  def rq_current_pos_norm(gripper_socket="1"):
      pos_gripper = rq_current_pos(gripper_socket)
      pos_norm = gripper_to_norm(pos_gripper)
      return pos_norm
  end

  def gripper_to_norm(value_gripper):
      value_norm = (value_gripper / 255) * 100
      return floor(value_norm)
  end

  def norm_to_gripper(value_norm):
      value_gripper = (value_norm / 100) * 255
      return ceil(value_gripper)
  end

  def rq_get_position():
      return rq_current_pos_norm()
  end

  def rq_gripper_led_on(gripper_socket="1"):
      rq_set_var("LBP",0, gripper_socket)
  end

  def rq_gripper_led_off(gripper_socket="1"):
      rq_set_var("LBP",1, gripper_socket)
      rq_set_var("LRD",0, gripper_socket)
      rq_set_var("LBL",0, gripper_socket)
      rq_set_var("LGN",0, gripper_socket)
  end

  def rq_gripper_led_force_red(gripper_socket="1"):
      rq_set_var("LBP",1, gripper_socket)
      rq_set_var("LRD",1, gripper_socket)
      rq_set_var("LBL",0, gripper_socket)
      rq_set_var("LGN",0, gripper_socket)
  end

  def rq_gripper_led_force_blue(gripper_socket="1"):
      rq_set_var("LBP",1, gripper_socket)
      rq_set_var("LRD",0, gripper_socket)
      rq_set_var("LBL",1, gripper_socket)
      rq_set_var("LGN",0, gripper_socket)
  end

  def rq_gripper_led_force_green(gripper_socket="1"):
      rq_set_var("LBP",1, gripper_socket)
      rq_set_var("LRD",0, gripper_socket)
      rq_set_var("LBL",0, gripper_socket)
      rq_set_var("LGN",1, gripper_socket)
  end

  def rq_gripper_led_force_purple(gripper_socket="1"):
      rq_set_var("LBP",1, gripper_socket)
      rq_set_var("LRD",1, gripper_socket)
      rq_set_var("LBL",1, gripper_socket)
      rq_set_var("LGN",0, gripper_socket)
  end

  ############################################
  # mm/inches functions
  ############################################
  gripper_closed_norm = [100, 100, 100, 100]
  gripper_open_norm = [0, 0, 0, 0]
  gripper_closed_mm = [0, 0, 0, 0]
  gripper_open_mm = [50, 50, 50, 50]

  def rq_current_pos_mm(gripper_socket=1):
      pos_gripper = rq_current_pos(gripper_socket)
      pos_mm = gripper_to_mm(pos_gripper, gripper_socket)
      return round_value_2_dec(pos_mm)
  end

  def rq_current_pos_inches(gripper_socket=1):
      pos_gripper = rq_current_pos(gripper_socket)
      pos_mm = gripper_to_mm(pos_gripper, gripper_socket)
      pos_in = pos_mm / 25.4
      return round_value_2_dec(pos_in)
  end

  def rq_move_mm(pos_mm, gripper_socket=1):
      pos_gripper = mm_to_gripper(pos_mm, gripper_socket)
      rq_move(pos_gripper, gripper_socket)
  end

  def rq_move_and_wait_mm(pos_mm, gripper_socket=1):
      pos_gripper = mm_to_gripper(pos_mm, gripper_socket)
      rq_move_and_wait(pos_gripper, gripper_socket)
  end

  def rq_move_inches(pos_in, gripper_socket=1):
      pos_mm = pos_in * 25.4
      rq_move_mm(pos_mm, gripper_socket)
  end

  def rq_move_and_wait_inches(pos_in, gripper_socket=1):
      pos_mm = pos_in * 25.4
      rq_move_and_wait_mm(pos_mm, gripper_socket)
  end

  def get_closed_norm(gripper_socket):
      return gripper_closed_norm[gripper_socket - 1]
  end

  def get_open_norm(gripper_socket):
      return gripper_open_norm[gripper_socket - 1]
  end

  def get_closed_mm(gripper_socket):
      return gripper_closed_mm[gripper_socket - 1]
  end

  def get_open_mm(gripper_socket):
      return gripper_open_mm[gripper_socket - 1]
  end

  def set_closed_norm(closed_norm, gripper_socket):
      gripper_closed_norm[gripper_socket - 1] = closed_norm
  end

  def set_open_norm(open_norm, gripper_socket):
      gripper_open_norm[gripper_socket - 1] = open_norm
  end

  def set_closed_mm(closed_mm, gripper_socket):
      gripper_closed_mm[gripper_socket - 1] = closed_mm
  end

  def set_open_mm(open_mm, gripper_socket):
      gripper_open_mm[gripper_socket - 1] = open_mm
  end

  def gripper_to_mm(value_gripper, gripper_socket):
      closed_norm = get_closed_norm(gripper_socket)
      open_norm = get_open_norm(gripper_socket)
      closed_mm = get_closed_mm(gripper_socket)
      open_mm = get_open_mm(gripper_socket)

      value_norm = (value_gripper / 255) * 100

      slope = (closed_mm - open_mm) / (closed_norm - open_norm)
      value_mm = slope * (value_norm - closed_norm) + closed_mm

      if (value_mm > open_mm):
          value_mm_limited = open_mm
      elif (value_mm < closed_mm):
          value_mm_limited = closed_mm
      else:
          value_mm_limited = value_mm
      end

      return value_mm_limited
  end

  def mm_to_gripper(value_mm, gripper_socket):
      closed_norm = get_closed_norm(gripper_socket)
      open_norm = get_open_norm(gripper_socket)
      closed_mm = get_closed_mm(gripper_socket)
      open_mm = get_open_mm(gripper_socket)

      slope = (closed_norm - open_norm) / (closed_mm - open_mm)
      value_norm = (value_mm - closed_mm) * slope + closed_norm

      value_gripper = value_norm * 255 / 100

      if (value_gripper > 255):
          value_gripper_limited = 255
      elif (value_gripper < 0):
          value_gripper_limited = 0
      else:
          value_gripper_limited = round_value(value_gripper)
      end

      return value_gripper_limited
  end

  def round_value(value):
      value_mod = value % 1

      if(value_mod < 0.5):
          return floor(value)
      else:
          return ceil(value)
      end
  end

  def round_value_2_dec(value):
      value_x_100 = value * 100
      value_x_100_rounded = round_value(value_x_100)
      return value_x_100_rounded / 100
  end

  def clear_socket_buffer(gripper_socket="1", read_timeout = 0.1):
      rq_comm_clear_socket_buffer_enabled[rq_socket_to_index(gripper_socket)] = True
  end

  def rq_gripper_id_to_ascii(gripper_id):
      if(gripper_id == "1"):
          return 57
      elif(gripper_id == "2"):
          return 50
      elif(gripper_id == "3"):
          return 51
      elif(gripper_id == "4"):
          return 52
      end
  end

  def scale(value, rawRange, scaledRange):
      def computeSlope(inputRange, outputRange):
          outputRangeDelta = outputRange[1] - outputRange[0]
          inputRangeDelta = inputRange[1] - inputRange[0]

          if (inputRangeDelta == 0):
              return 0
          else:
              return outputRangeDelta / inputRangeDelta
          end
      end

      def computeIntercept(slope, inputRange, outputRange):
          return outputRange[0] - (slope * inputRange[0])
      end

      def clipScaledValue(outputScaledValue, outputRange):
          if (outputRange[0] < outputRange[1]):
              return clipWhenLowerLimitIsLessThanHigher(outputScaledValue, outputRange)
          else:
              return clipWhenLowerLimitIsGreaterThanHigherLimit(outputScaledValue, outputRange)
          end
      end

      def clipWhenLowerLimitIsGreaterThanHigherLimit(outputScaledValue, outputRange):
          if (outputScaledValue < outputRange[1]):
              return outputRange[1]
          elif (outputScaledValue > outputRange[0]):
              return outputRange[0]
          else:
              return outputScaledValue
          end
      end

      def clipWhenLowerLimitIsLessThanHigher(outputScaledValue, outputRange):
          if (outputScaledValue < outputRange[0]):
              return outputRange[0]
          elif (outputScaledValue > outputRange[1]):
              return outputRange[1]
          else:
              return outputScaledValue
          end
      end

      slope = computeSlope(rawRange, scaledRange)
      intercept = computeIntercept(slope, rawRange, scaledRange)
      scaledValue = slope * value + intercept
      return clipScaledValue(scaledValue, scaledRange)
  end

  def limit(value, range):
      return scale(value, range, range)
  end


  rq_init_comm_if_connected(9, "1")
  rq_init_comm_if_connected(2, "2")
  rq_init_comm_if_connected(3, "3")
  rq_init_comm_if_connected(4, "4")
  rq_print_connected_grippers()
  rq_gripper_communication_thread = run rq_gripper_communication()
  set_closed_norm(100.0, 1)
  set_open_norm(0.0, 1)
  set_closed_mm(0.0, 1)
  set_open_mm(50.0, 1)
  set_closed_norm(100.0, 2)
  set_open_norm(0.0, 2)
  set_closed_mm(0.0, 2)
  set_open_mm(50.0, 2)
  set_closed_norm(100.0, 3)
  set_open_norm(0.0, 3)
  set_closed_mm(0.0, 3)
  set_open_mm(50.0, 3)
  set_closed_norm(100.0, 4)
  set_open_norm(0.0, 4)
  set_closed_mm(0.0, 4)
  set_open_mm(50.0, 4)
  rq_current_limit_enabled = False
  while(not rq_gripper_communication_thread_started):
      sleep(0.008)
  end
  # end: URCap Installation Node
  global cnt_1=0
  global volo=0
  global volo_is_counting=False
  thread Timer_Thread():
    while (True):
      if (volo_is_counting):
        volo = volo + get_steptime()
      end
      sync()
    end
  end
  run Timer_Thread()
  while (True):
    $ 1 "Robot Program"
    # begin: URCap Program Node
    #   Source: Robotiq_Grippers, 1.8.9.14887, Robotiq Inc.
    #   Type: Gripper Activate
    $ 2 "Gripper Activate"

    kill rq_gripper_communication_thread
    rq_gripper_communication_thread_started = False
    rq_close_gripper_socket("1")
    rq_close_gripper_socket("2")
    rq_close_gripper_socket("3")
    rq_close_gripper_socket("4")

    rq_init_comm_if_connected(9, "1")
    rq_init_comm_if_connected(2, "2")
    rq_init_comm_if_connected(3, "3")
    rq_init_comm_if_connected(4, "4")
    rq_print_connected_grippers()
    rq_gripper_communication_thread = run rq_gripper_communication()

    while(not rq_gripper_communication_thread_started):
        sleep(0.008)
    end

    rq_set_max_current_for_all_grippers()

    reset_and_activate = False

    rq_activate_all_grippers(False)
    # end: URCap Program Node
    # begin: URCap Program Node
    #   Source: Robotiq_Grippers, 1.8.9.14887, Robotiq Inc.
    #   Type: Gripper
    $ 3 "Gripper Open (1)"
    if not(gripper_connected[0]):
      popup("Gripper 1 must be connected to run this program.", "No connection", False, True, True)
    end
    if not(rq_is_gripper_activated("1")):
      popup("Gripper 1 is not activated. Go to Installation tab > Gripper to activate it and run the program again.", "Not activated", False, True, True)
    end
    rq_set_pos_spd_for(0, 0, 0, "1")
    rq_wait_pos_spe_for_request(0, 0, 0, "1")
    rq_go_to("1")
    rq_wait("1")
    # end: URCap Program Node
    $ 4 "volo: Stop"
    volo_is_counting = False
    $ 5 "ready≔ False "
    global ready=  False
    $ 6 "engineon≔Nastro_ON"
    global engineon=get_standard_digital_out(0)
    $ 7 "engineon≔ False "
    global engineon=  False
    $ 8 "sensoreBasso≔FC_Start"
    global sensoreBasso=get_standard_digital_in(4)
    $ 9 "sensoreAlto≔FC_High"
    global sensoreAlto=get_standard_digital_in(6)
    $ 10 "sensoreStop≔FC_End"
    global sensoreStop=get_standard_digital_in(5)
    $ 11 "tempoVolo≔4000"
    global tempoVolo=4000
    $ 12 "Loop"
    while (True):
      $ 13 "If FC_Start== True "
      if (get_standard_digital_in(4)==  True  ):
        $ 14 "engineon≔ True "
        global engineon=  True
        $ 15 "Wait FC_Start=LO"
        while (get_standard_digital_in(4) == True):
          sync()
        end
      else:
        $ 16 "ElseIf FC_High== True "
        if (get_standard_digital_in(6)==  True  ):
          $ 17 "engineon≔ True "
          global engineon=  True
          $ 18 "Wait FC_High=LO"
          while (get_standard_digital_in(6) == True):
            sync()
          end
        else:
          $ 19 "ElseIf FC_End== True "
          if (get_standard_digital_in(5)==  True  ):
            $ 20 "engineon≔ False "
            global engineon=  False
            $ 21 "MoveL"
            $ 22 "Waypoint_1" "breakAfter"
            movel(p[-.381387685375, -.169307009528, .186364165479, .031229211360, 3.092074785863, -.049669567106], a=1.2, v=0.25)
            $ 23 "MoveL"
            $ 24 "Waypoint_2" "breakAfter"
            movel(p[-.373641097354, -.171322588210, .081624890856, .031253673923, 3.092083063402, -.049651173659], a=1.2, v=0.25)
            # begin: URCap Program Node
            #   Source: Robotiq_Grippers, 1.8.9.14887, Robotiq Inc.
            #   Type: Gripper
            $ 25 "Gripper Move51% (1)"
            if not(gripper_connected[0]):
              popup("Gripper 1 must be connected to run this program.", "No connection", False, True, True)
            end
            if not(rq_is_gripper_activated("1")):
              popup("Gripper 1 is not activated. Go to Installation tab > Gripper to activate it and run the program again.", "Not activated", False, True, True)
            end
            rq_set_pos_spd_for(131, 0, 0, "1")
            rq_wait_pos_spe_for_request(131, 0, 0, "1")
            rq_go_to("1")
            rq_wait("1")
            # end: URCap Program Node
            $ 26 "MoveL"
            $ 27 "Waypoint_3" "breakAfter"
            movel(p[-.370356696043, -.174547637783, .216862429798, .031961409927, 3.097477882431, -.043978030525], a=1.2, v=0.25)
            $ 28 "MoveL"
            $ 29 "Waypoint_4" "breakAfter"
            movel(p[-.134875456305, -.252278271452, .221726537061, .032070337176, 3.097477750080, -.043854214395], a=1.2, v=0.25)
            $ 30 "Pallet"
            cnt_1_x = cnt_1 % 2
            cnt_1_y = floor(cnt_1 / 2)
            pose_1 = interpolate_pose(interpolate_pose(p[-.089762363593, -.429151138960, .009188706301, .027577147014, 3.053416589493, -.032182313128], p[.031186609987, -.429171211043, .011085502208, .027611575133, 3.053453182137, -.032263865590], cnt_1_x/1), interpolate_pose(p[-.089761553552, -.366553516844, .009168617974, .027481938487, 3.053493094310, -.032138841944], p[.031156149702, -.364086955268, .011056827590, .027631286382, 3.053463713793, -.032250855705],cnt_1_x/1), cnt_1_y/1)
            if (cnt_1 >= 3):
              cnt_1 = 0
            else:
              cnt_1 = cnt_1 + 1
            end
            $ 37 "Approach_1" "noBreak"
            movel(pose_trans(pose_1, pose_trans(pose_inv(p[-.089755279794, -.366542025468, .202492381968, .027482330613, 3.053431155792, -.032206448903]),p[-.089781181398, -.366546626212, .202507837739, .027606886294, 3.053463920443, -.032300040654])), a=1.2, v=0.25)
            $ 38 "PatternPoint_1" "noBreak"
            movel(pose_1, a=1.2, v=0.25)
            $ 39 "Set" "noBreak"
            $ 40 "Wait volo>tempoVolo" "noBreak"
            while (not(volo>tempoVolo)):
              sync()
            end
            $ 41 "Exit_1" "noBreak"
            movel(pose_trans(pose_1, pose_trans(pose_inv(p[-.089755279794, -.366542025468, .202492381968, .027482330613, 3.053431155792, -.032206448903]),p[-.089763731108, -.366543702749, .202497776555, .027500770851, 3.053466015947, -.032225658991])), a=1.2, v=0.25)
            $ 42 "volo: Start"
            volo_is_counting = True
            $ 43 "volo: Reset"
            volo = 0
          else:
            $ 44 "ElseIf volo>tempoVolo"
            if (volo>tempoVolo):
              $ 45 "volo: Stop"
              volo_is_counting = False
              $ 46 "volo: Reset"
              volo = 0
            end
          end
        end
      end
    end
  end
end
